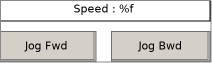
VISUALIZATION Conveyor  // 212x63
VAR_IN_OUT
	bJogFwd: BOOL;
	bJogBwd: BOOL;
	fSpeed: LREAL;
END_VAR
    Rectangle (-3,-3 213x24), "Speed : %f", text variable: fSpeed
    Button (-3,31 99x30), "Jog Fwd"
        tap bJogFwd
    Button (111,31 99x30), "Jog Bwd"
        tap bJogBwd
END_VISUALIZATION

(* stored: Version 1.1.0.1
   Visu Conveyor: Id {f89cd03f-2968-404b-ab35-09de65a27c07} *)
